// Mitsubishi GX Works2 project: Sugmaskin   PLC: FX1S

// global labels: Global1
VAR_GLOBAL
  SUGKOPP_UPPE AT X001 : BOOL;
  SUGKOPP_NERE AT X002 : BOOL;
  SUGKOPP_VÄNSTER AT X003 : BOOL;
  SUGKOPP_HÖGER AT X004 : BOOL;
  SUG_UPPNÅTT AT X005 : BOOL;
  SLÄDE_VÄNSTER AT X006 : BOOL;
  SLÄDE_HÖGER AT X007 : BOOL;
  SUGROTOR_MOTSOLS AT Y000 : BOOL;
  SUGROTOR_MEDSOLS AT Y001 : BOOL;
  SUGKOLV_NER AT Y002 : BOOL;
  SLÄDE_GÅ_HÖGER AT Y003 : BOOL;
  SLÄDE_GÅ_VÄNSTER AT Y004 : BOOL;
  SUGEJEKTOR AT Y005 : BOOL;
  INIT_PULS AT M8002 : BOOL;
  STEG_1 AT M1 : BOOL;
  STEG_2 AT M2 : BOOL;
  STEG_3 AT M3 : BOOL;
  STEG_4 AT M4 : BOOL;
  STEG_5 AT M5 : BOOL;
  STEG_6 AT M6 : BOOL;
  STEG_7 AT M7 : BOOL;
  STEG_8 AT M8 : BOOL;
  STEG_9 AT M9 : BOOL;
  STEG_10 AT M10 : BOOL;
  SUG_EJ_UPPNÅTT AT M11 : BOOL;
  START_RESET AT X000 : BOOL;
  RESETMINNE AT M12 : BOOL;
  RÄKNARMINNE AT M13 : BOOL;
END_VAR

// task Task_01 (event TRUE, interval 0, priority 31): Ladder, Aktivation

PROGRAM Ladder
VAR
  Nada : BOOL;
  SugTimer : INT;
END_VAR
(* structured ladder/FBD written out as ST: instructions are called as NAME(EN, inputs, outputs); _pN, _eN, _tN stand for wires *)
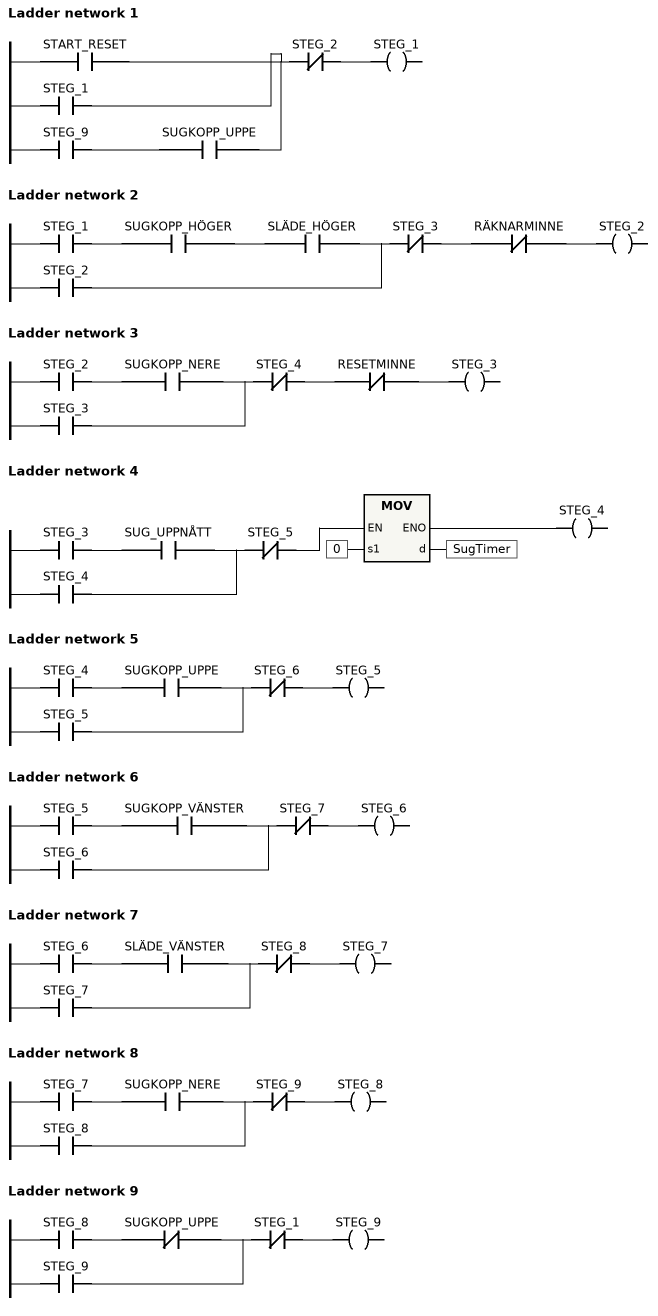
(* network 1 *)
STEG_1 := (START_RESET OR STEG_1 OR (STEG_9 AND SUGKOPP_UPPE)) AND NOT STEG_2;
(* network 2 *)
STEG_2 := (((STEG_1 AND SUGKOPP_HÖGER AND SLÄDE_HÖGER) OR STEG_2) AND NOT STEG_3) AND NOT RÄKNARMINNE;
(* network 3 *)
STEG_3 := (((STEG_2 AND SUGKOPP_NERE) OR STEG_3) AND NOT STEG_4) AND NOT RESETMINNE;
(* network 4 *)
_e1 := MOV(((STEG_3 AND SUG_UPPNÅTT) OR STEG_4) AND NOT STEG_5, 0, SugTimer);
STEG_4 := _e1;
(* network 5 *)
STEG_5 := ((STEG_4 AND SUGKOPP_UPPE) OR STEG_5) AND NOT STEG_6;
(* network 6 *)
STEG_6 := ((STEG_5 AND SUGKOPP_VÄNSTER) OR STEG_6) AND NOT STEG_7;
(* network 7 *)
STEG_7 := ((STEG_6 AND SLÄDE_VÄNSTER) OR STEG_7) AND NOT STEG_8;
(* network 8 *)
STEG_8 := ((STEG_7 AND SUGKOPP_NERE) OR STEG_8) AND NOT STEG_9;
(* network 9 *)
STEG_9 := ((STEG_8 AND NOT SUGKOPP_UPPE) OR STEG_9) AND NOT STEG_1;
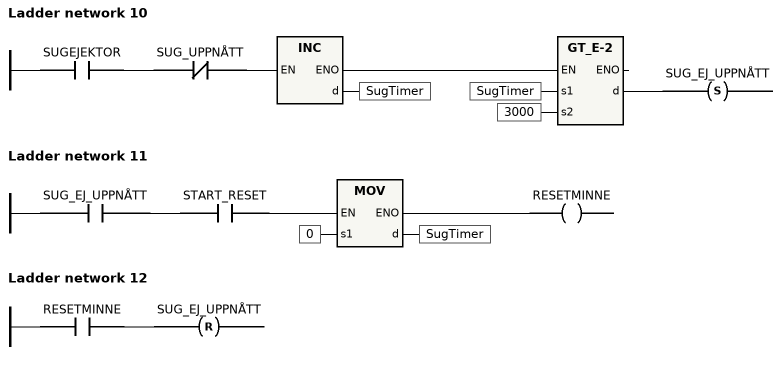
(* network 10 *)
_e1 := INC(SUGEJEKTOR AND NOT SUG_UPPNÅTT, SugTimer);
GT_E(_e1, SugTimer, 3000, _t2);
SET(_t2, SUG_EJ_UPPNÅTT);
(* network 11 *)
_e1 := MOV(SUG_EJ_UPPNÅTT AND START_RESET, 0, SugTimer);
RESETMINNE := _e1;
(* network 12 *)
RST(RESETMINNE, SUG_EJ_UPPNÅTT);
END_PROGRAM

PROGRAM Aktivation
(* structured ladder/FBD written out as ST: instructions are called as NAME(EN, inputs, outputs); _pN, _eN, _tN stand for wires *)
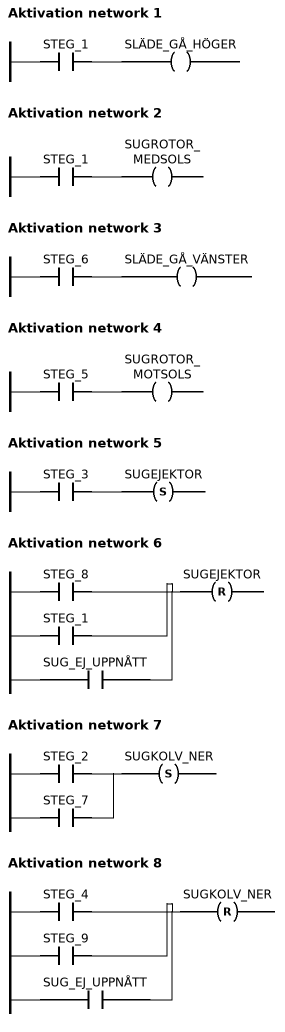
(* network 1 *)
SLÄDE_GÅ_HÖGER := STEG_1;
(* network 2 *)
SUGROTOR_MEDSOLS := STEG_1;
(* network 3 *)
SLÄDE_GÅ_VÄNSTER := STEG_6;
(* network 4 *)
SUGROTOR_MOTSOLS := STEG_5;
(* network 5 *)
SET(STEG_3, SUGEJEKTOR);
(* network 6 *)
RST(STEG_8 OR STEG_1 OR SUG_EJ_UPPNÅTT, SUGEJEKTOR);
(* network 7 *)
SET(STEG_2 OR STEG_7, SUGKOLV_NER);
(* network 8 *)
RST(STEG_4 OR STEG_9 OR SUG_EJ_UPPNÅTT, SUGKOLV_NER);
END_PROGRAM
